(* PLC project STD_TEST, LOLITECH BREMIZ 1 *)
(* stored: companyURL www.lolitech.com, productRelease 1, creationDateTime 2007-07-07 11:58:26, contentDescription This tests as most as possible IEC standard library, modificationDateTime 2008-08-27 16:29:04 *)

TYPE MYTYPE : INT(0..1000);
END_TYPE

TYPE MYTYPE2 : (OPEN, CLOSED) := CLOSED;
END_TYPE

TYPE MYTYPE3 : ARRAY[1..8, 1..8] OF MYTYPE5 := [32(0), 30(1)];
END_TYPE

TYPE MYTYPE4 : UINT(1..100);
END_TYPE

TYPE MYTYPE5 : MYTYPE4 := 10;
END_TYPE

FUNCTION_BLOCK Bitwise_Block
  VAR_INPUT
    IN1 : BOOL;
    IN2 : BOOL;
  END_VAR
  VAR_OUTPUT
    OUT_AND : BOOL;
    OUT_OR : BOOL;
    OUT_XOR : BOOL;
    OUT_SR : BOOL;
  END_VAR
  VAR
    SR1 : SR;
  END_VAR

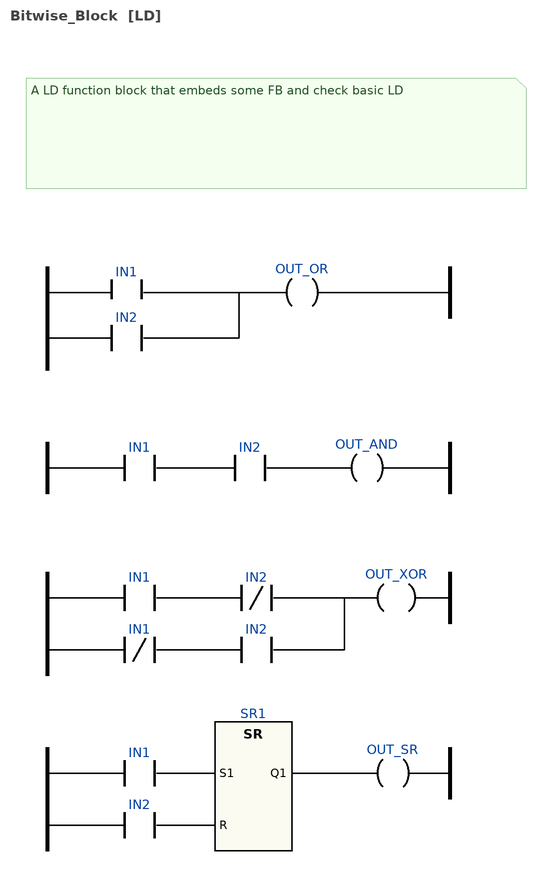
(* LD diagram, written out as Structured Text *)
(* A LD function block that embeds some FB and check basic LD *)
OUT_OR := IN1 OR IN2;
OUT_AND := IN1 AND IN2;
OUT_XOR := IN1 AND NOT IN2 OR NOT IN1 AND IN2;
SR1(S1 := IN1, R := IN2);
OUT_SR := SR1.Q1;
END_FUNCTION_BLOCK

FUNCTION GETBIT : BOOL
  VAR_INPUT
    INPUT_BYTE : BYTE;
    NUM_BIT : USINT;
  END_VAR

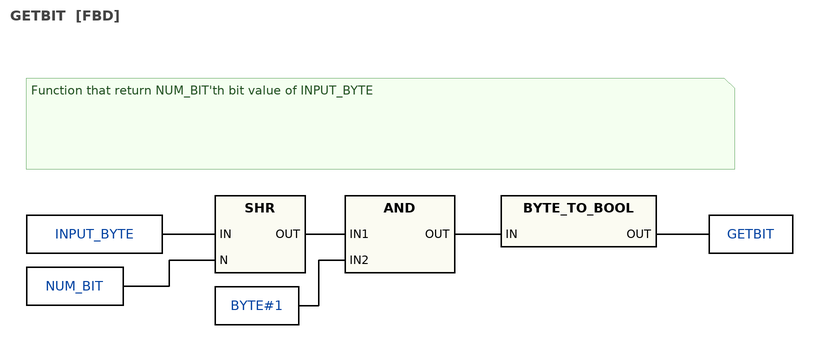
(* FBD diagram, written out as Structured Text *)
(* Function that return NUM_BIT'th bit value of INPUT_BYTE *)
GETBIT := BYTE_TO_BOOL(SHR(INPUT_BYTE, NUM_BIT) AND BYTE#1);
END_FUNCTION

FUNCTION SETBIT : BYTE
  VAR_INPUT
    INPUT_BYTE : BYTE;
    INPUT_BIT : BOOL;
    NUM_BIT : USINT;
  END_VAR

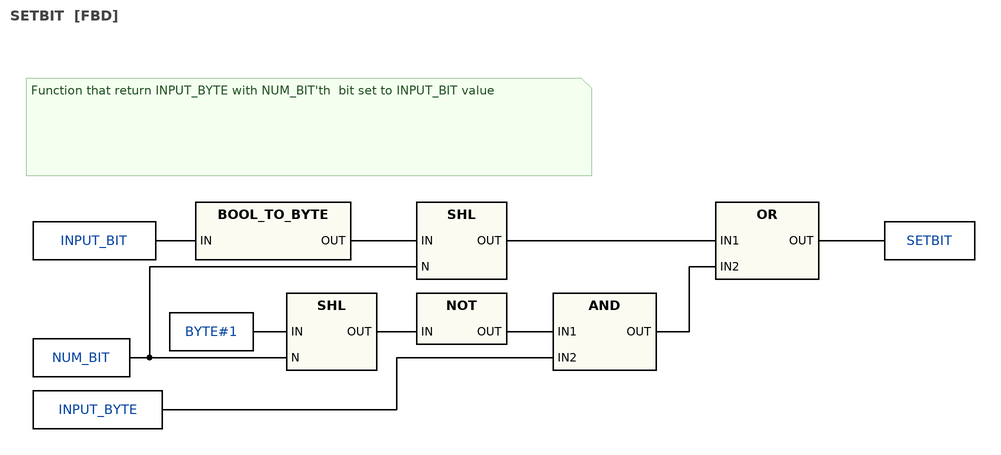
(* FBD diagram, written out as Structured Text *)
(* Function that return INPUT_BYTE with NUM_BIT'th  bit set to INPUT_BIT value *)
SETBIT := SHL(BOOL_TO_BYTE(INPUT_BIT), NUM_BIT) OR NOT SHL(BYTE#1, NUM_BIT) AND INPUT_BYTE;
END_FUNCTION

FUNCTION_BLOCK Test_SFC
  VAR_INPUT
    CNT1 : BOOL;
    CNT2 : BOOL;
    IN1 : MYTYPE;
    IN2 : MYTYPE;
    UPPER1 : INT;
    UPPER2 : INT;
  END_VAR
  VAR_OUTPUT
    OUT1 : MYTYPE;
    OUT2 : MYTYPE;
  END_VAR
  VAR
    TEST_ENUM : MYTYPE2;
    TEST_ARRAY : MYTYPE3;
  END_VAR
  VAR  (* added by the conversion: wires and edge detectors of the diagram *)
    _AND34_OUT : BOOL;
  END_VAR

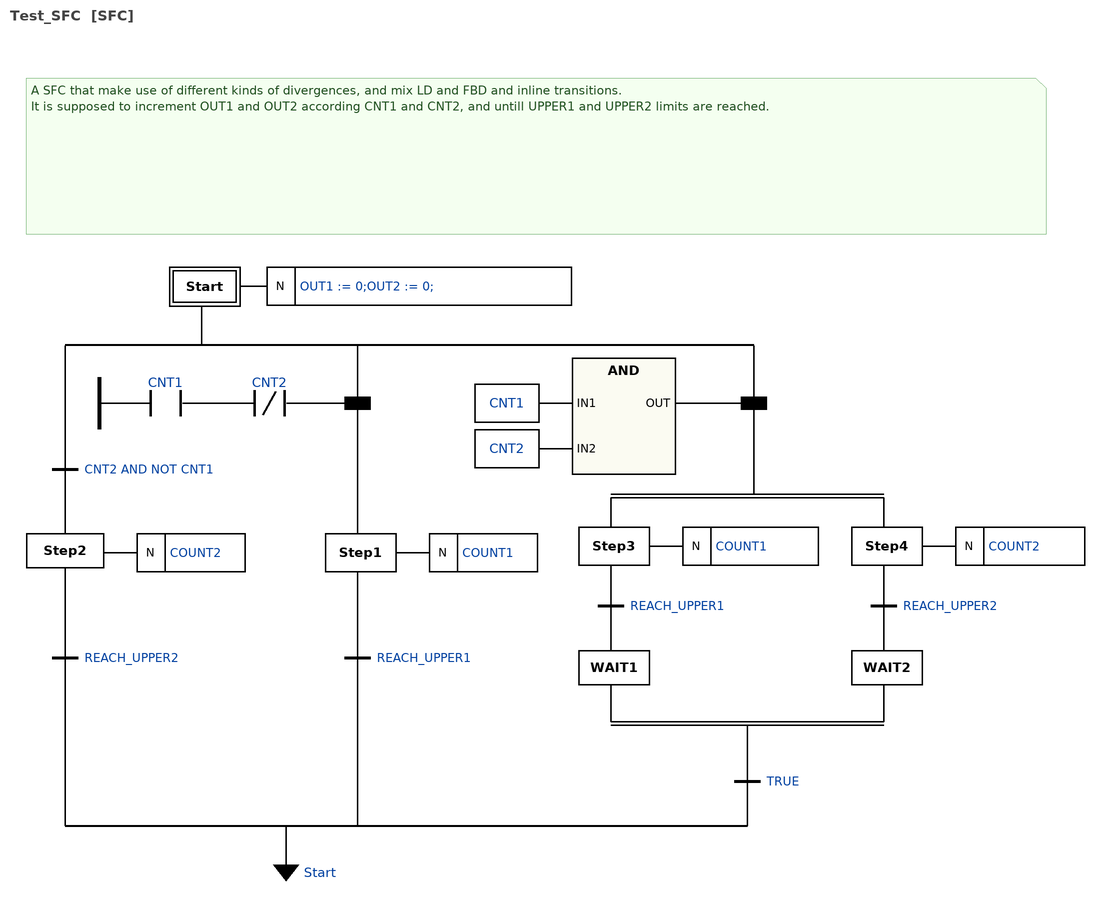
(* A SFC that make use of different kinds of divergences, and mix LD and FBD and inline transitions.
It is supposed to increment OUT1 and OUT2 according CNT1 and CNT2, and untill UPPER1 and UPPER2 limits are reached. *)
INITIAL_STEP Start:
  START_INLINE1(N);
  COMPUTE_FUNCTION_BLOCKS(S);
END_STEP
ACTION START_INLINE1:
  OUT1 := 0;OUT2 := 0;
END_ACTION
TRANSITION FROM Start TO Step2
  := CNT2 AND NOT CNT1;
END_TRANSITION
TRANSITION FROM Start TO Step1
  := CNT1 AND NOT CNT2;
END_TRANSITION
TRANSITION FROM Start TO (Step3, Step4)
  := _AND34_OUT;
END_TRANSITION
STEP Step3:
  COUNT1(N);
END_STEP
TRANSITION FROM Step3 TO WAIT1  (* REACH_UPPER1 *)
  := OUT1 >= UPPER1;
END_TRANSITION
STEP Step4:
  COUNT2(N);
END_STEP
TRANSITION FROM Step4 TO WAIT2  (* REACH_UPPER2 *)
  := OUT2 >= UPPER2;
END_TRANSITION
STEP Step2:
  COUNT2(N);
END_STEP
TRANSITION FROM Step2 TO Start  (* REACH_UPPER2 *)
  := OUT2 >= UPPER2;
END_TRANSITION
STEP Step1:
  COUNT1(N);
END_STEP
TRANSITION FROM Step1 TO Start  (* REACH_UPPER1 *)
  := OUT1 >= UPPER1;
END_TRANSITION
STEP WAIT1:
END_STEP
TRANSITION FROM (WAIT1, WAIT2) TO Start
  := TRUE;
END_TRANSITION
STEP WAIT2:
END_STEP
ACTION COMPUTE_FUNCTION_BLOCKS:  (* blocks drawn on the SFC sheet *)
  _AND34_OUT := CNT1 AND CNT2;
END_ACTION

ACTION COUNT1:
OUT1 := IN1 + 1;
TEST_ENUM := OPEN;

              
END_ACTION

ACTION COUNT2:
OUT2 := IN2 + 1;
TEST_ARRAY[0,0] := TEST_ARRAY[0,1] + 50;

              
END_ACTION
END_FUNCTION_BLOCK

PROGRAM MAIN_TEST
  VAR
    DigitalOut AT %QB0.0.16.25088.1 : BYTE;
    DigitalIn AT %IB0.0.32.24576.1 : BYTE;
    AnalogOut1 AT %QW0.0.16.25617.1 : MYTYPE;
    AnalogOut2 AT %QW0.0.16.25617.2 : MYTYPE;
    AnalogOut3 AT %QW0.0.16.25617.3 : INT;
    AnalogIn1 AT %IW0.0.32.25601.1 : INT;
    AnalogIn2 AT %IW0.0.32.25601.2 : INT;
  END_VAR
  VAR
    Test : Bitwise_Block;
    Test2 : Test_SFC;
    t1 : TOF;
    latch : RS;
    t2 : TOF;
  END_VAR
  VAR  (* added by the conversion: wires and edge detectors of the diagram *)
    _GETBIT37_OUT : BOOL;
    _GETBIT44_OUT : BOOL;
  END_VAR

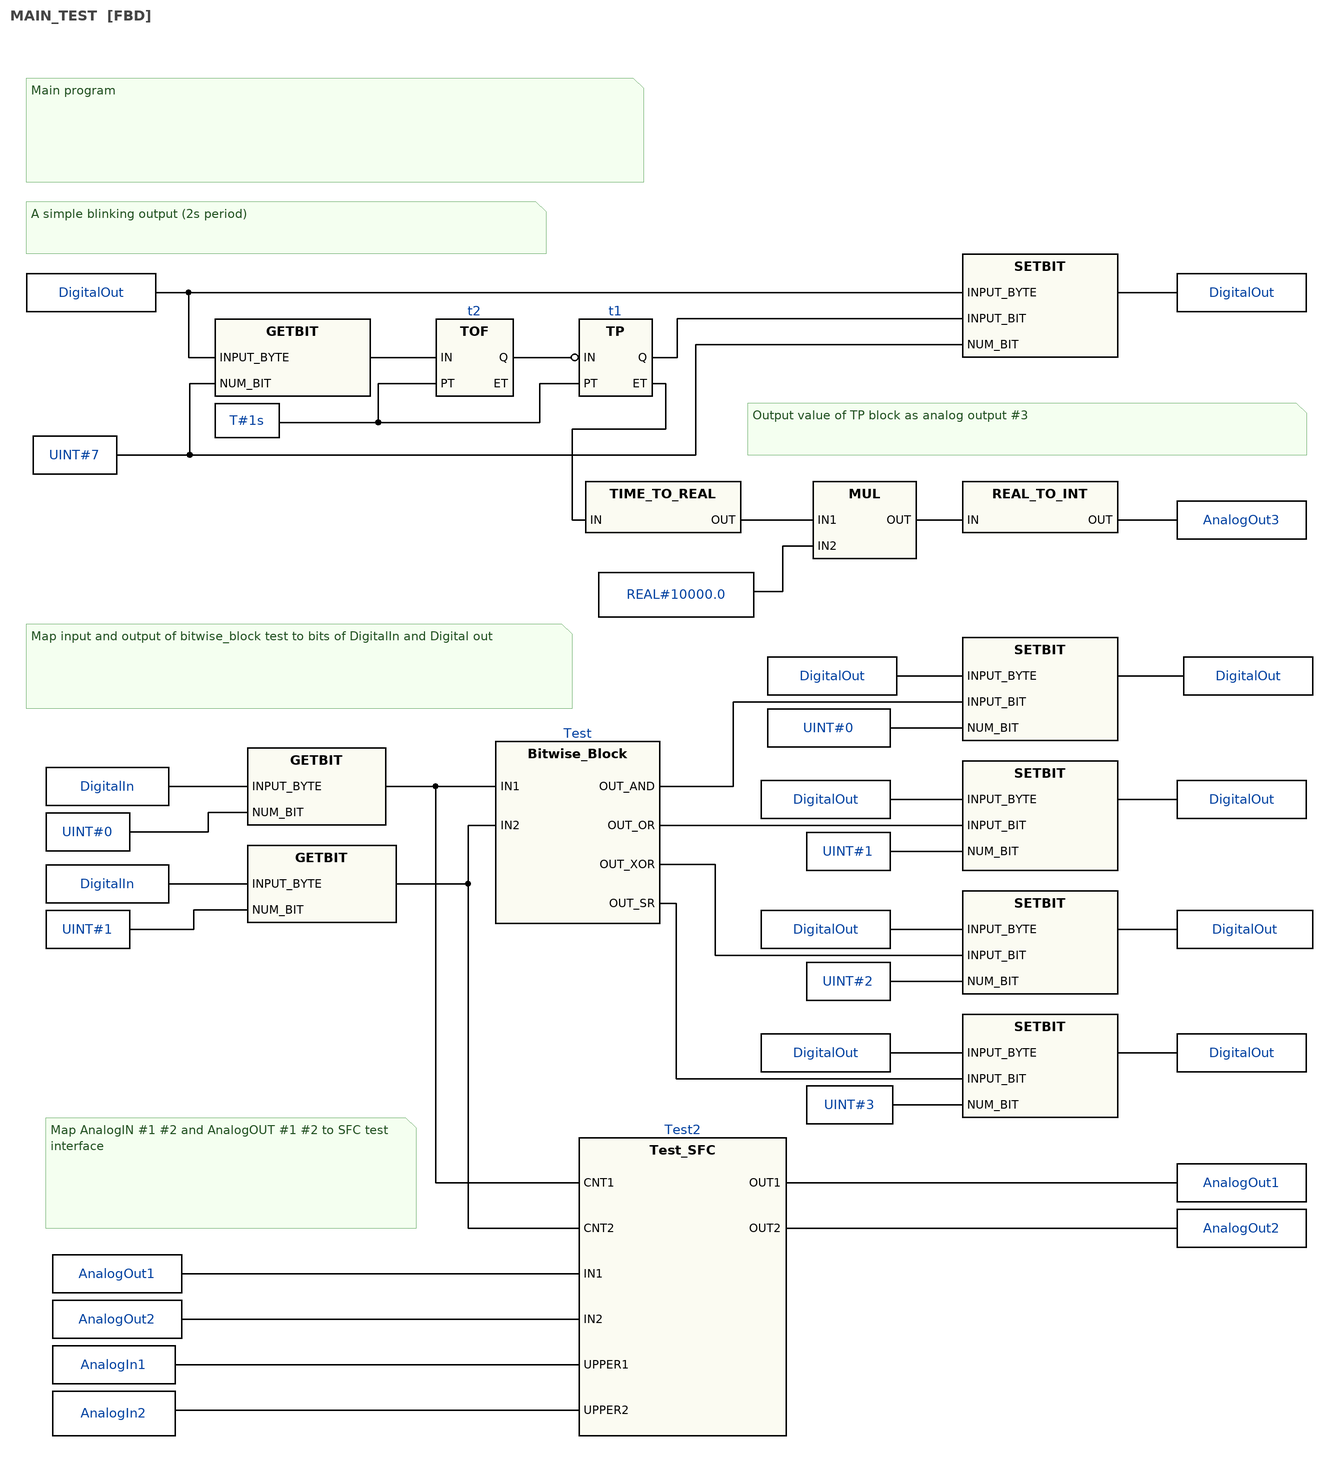
(* FBD diagram, written out as Structured Text *)
(* Main program *)
(* A simple blinking output (2s period) *)
t2(IN := GETBIT(DigitalOut, UINT#7), PT := T#1s);
t1(IN := NOT t2.Q, PT := T#1s);
DigitalOut := SETBIT(DigitalOut, t1.Q, UINT#7);
(* Output value of TP block as analog output #3 *)
AnalogOut3 := REAL_TO_INT(TIME_TO_REAL(t1.ET) * REAL#10000.0);
(* Map input and output of bitwise_block test to bits of DigitalIn and Digital out *)
_GETBIT37_OUT := GETBIT(DigitalIn, UINT#0);
_GETBIT44_OUT := GETBIT(DigitalIn, UINT#1);
Test(IN1 := _GETBIT37_OUT, IN2 := _GETBIT44_OUT);
DigitalOut := SETBIT(DigitalOut, Test.OUT_AND, UINT#0);
DigitalOut := SETBIT(DigitalOut, Test.OUT_OR, UINT#1);
DigitalOut := SETBIT(DigitalOut, Test.OUT_XOR, UINT#2);
DigitalOut := SETBIT(DigitalOut, Test.OUT_SR, UINT#3);
(* Map AnalogIN #1 #2 and AnalogOUT #1 #2 to SFC test interface *)
Test2(CNT1 := _GETBIT37_OUT, CNT2 := _GETBIT44_OUT, IN1 := AnalogOut1, IN2 := AnalogOut2, UPPER1 := AnalogIn1, UPPER2 := AnalogIn2);
AnalogOut1 := Test2.OUT1;
AnalogOut2 := Test2.OUT2;
END_PROGRAM

CONFIGURATION STD_CONF
  RESOURCE STD_RESSOURCE ON PLC
    TASK STD_TASK(INTERVAL := 00:00:00.100000, PRIORITY := 0);
    PROGRAM MAIN_INSTANCE WITH STD_TASK : MAIN_TEST;
  END_RESOURCE
END_CONFIGURATION
